Universal Robots PolyScope program: open.urp

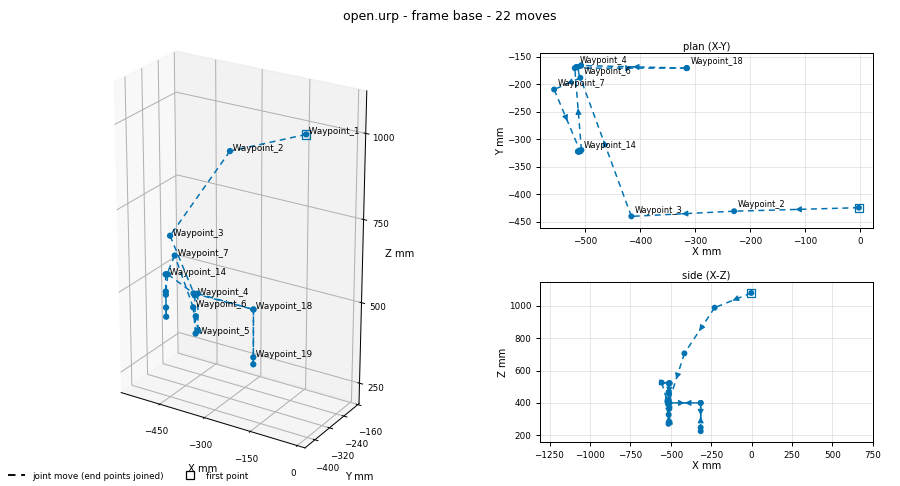
[picture p0: tool path of open.urp in frame base, 22 of 22 moves have a stored position in this frame; points joined in program order, loops and branches not executed]
Program open (installation=default directory=/programs/PrakjoyShi_Beer createdIn=5.12.6.1102099 lastSavedIn=5.12.6.1102099 robotSerialNumber=20215500597)
Calibrated DH parameters: a=[0.000193, -0.066673, -0.391568, -0.000012, 0.00005, 0]; d=[0.162643, -472.05677, 465.132521, 7.058239, 0.099746, 0.099582]; alpha=[1.571116, 0.00089, 0.003862, 1.569269, -1.569248, 0]; deltaTheta=[0, -1.413394, 7.628392, 0.068187, 0, -0.000001]
Robot Program (runOnlyOnce=true)
  MoveJ speed 60 deg/s, acceleration 80 deg/s^2 (useActiveTCP=true) feature=Base
    Waypoint Waypoint_1: TCP in base x=-1.583 y=-424.817 z=1080.554 mm, rx=-0.0045 ry=-2.2185 rz=2.2204 rad; joints [0.002, -89.999, 0.003, -90.001, -0.003, 0.002] deg; TCP offset x=0 y=0 z=191.5 mm, rx=0 ry=0 rz=0 rad
    Waypoint Waypoint_2: TCP in base x=-228.579 y=-431.222 z=989.425 mm, rx=0.1477 ry=-2.1757 rz=2.1747 rad; joints [1.493, -89.92, 39.368, -135.847, 0.07, 0.005] deg
    Waypoint Waypoint_3: TCP in base x=-415.572 y=-440.598 z=706.538 mm, rx=0.0374 ry=2.1727 rz=-2.163 rad; joints [2.063, -85.755, 82.589, -172.267, 0.054, -0.516] deg
    Waypoint Waypoint_4: TCP in base x=-515.642 y=-168.639 z=393.174 mm, rx=-2.1836 ry=-2.2574 rz=0.0027 rad; joints [3.827, -83.832, 69.203, -75.39, -89.793, 1.925] deg
    URCap Gripper Activate (Robotiq_Grippers, Robotiq Inc.) dataModel(ResetAndActivateKey=false)
    URCap Gripper (Robotiq_Grippers, Robotiq Inc.) dataModel(position=0.0, force=63.92156862745098, speed=100.0, positionInDouble=0.0, forceInDouble=63.92156862745098, speedInDouble=100.0, slaveIds=[9], blocking=true)
    Waypoint Waypoint_5: TCP in base x=-513.995 y=-168.756 z=271.062 mm, rx=-2.1837 ry=-2.2577 rz=0.0027 rad; joints [3.824, -85.645, 89.178, -93.541, -89.77, 1.988] deg
  URCap Gripper (Robotiq_Grippers, Robotiq Inc.) dataModel(position=38.0, force=100.0, speed=100.0, positionInDouble=38.0, forceInDouble=100.0, speedInDouble=100.0, slaveIds=[9], blocking=true)
  MoveJ speed 60 deg/s, acceleration 80 deg/s^2 (useActiveTCP=true) feature=Base
    Waypoint Waypoint_6: TCP in base x=-508.355 y=-188.557 z=365.162 mm, rx=2.1753 ry=2.2666 rz=0 rad; joints [6.069, -84.648, 74.27, -79.533, -89.815, 3.731] deg
    Waypoint Waypoint_7: TCP in base x=-556.081 y=-209.772 z=525.944 mm, rx=-2.4486 ry=-1.9682 rz=0.0001 rad; joints [7.701, -60.708, 14.386, -43.591, -89.88, 20.001] deg
    Waypoint Waypoint_14: TCP in base x=-508.478 y=-322.557 z=521.579 mm, rx=-2.2014 ry=-2.2234 rz=0.0401 rad; joints [19.595, -63.115, 20.022, -48.453, -89.874, 18.926] deg
    Waypoint Waypoint_15: TCP in base x=-512.267 y=-322.567 z=521.57 mm, rx=-2.2014 ry=-2.2234 rz=0.0401 rad; joints [19.472, -62.139, 18.378, -47.783, -89.873, 18.801] deg
    Waypoint Waypoint_11: TCP in base x=-512.289 y=-322.554 z=458.084 mm, rx=-2.2014 ry=-2.2234 rz=0.0402 rad; joints [19.456, -71.678, 44.329, -64.2, -89.837, 18.84] deg
    Waypoint Waypoint_16: TCP in base x=-512.283 y=-322.575 z=417.932 mm, rx=-2.2013 ry=-2.2234 rz=0.0402 rad; joints [19.451, -74.525, 54.555, -71.58, -89.828, 18.862] deg
    Waypoint Waypoint_8: TCP in base x=-512.296 y=-322.578 z=389.017 mm, rx=-2.2014 ry=-2.2233 rz=0.0403 rad; joints [19.444, -75.91, 60.769, -76.41, -89.819, 18.877] deg
    Waypoint Waypoint_17: TCP in base x=-512.289 y=-322.57 z=468.034 mm, rx=-2.2014 ry=-2.2234 rz=0.0402 rad; joints [19.46, -70.742, 41.373, -62.179, -89.843, 18.837] deg
    Waypoint Waypoint_9: TCP in base x=-506.421 y=-319.932 z=522.217 mm, rx=-2.188 ry=-2.2544 rz=0.0003 rad; joints [19.417, -60.379, 14.59, -44.133, -89.874, 17.591] deg; TCP offset x=0 y=0 z=191.5 mm, rx=0 ry=0 rz=0 rad
    Waypoint Waypoint_10: TCP in base x=-518.545 y=-170.891 z=400.25 mm, rx=2.2171 ry=2.2233 rz=-0.0042 rad; joints [3.97, -83.045, 67.23, -74.144, -89.646, 3.807] deg; TCP offset x=0 y=0 z=191.5 mm, rx=0 ry=0 rz=0 rad
    Waypoint Waypoint_18: TCP in base x=-314.832 y=-170.884 z=400.234 mm, rx=2.2171 ry=2.2233 rz=-0.0041 rad; joints [6.401, -109.126, 90.204, -71.044, -89.654, 6.252] deg
    Waypoint Waypoint_19: TCP in base x=-314.834 y=-170.918 z=247.923 mm, rx=2.217 ry=2.2233 rz=-0.0042 rad; joints [6.362, -112.11, 114.622, -92.479, -89.633, 6.291] deg
    Waypoint Waypoint_20: TCP in base x=-314.83 y=-170.903 z=225.152 mm, rx=2.217 ry=2.2233 rz=-0.0043 rad; joints [6.354, -111.859, 117.807, -95.918, -89.633, 6.297] deg
    Waypoint Waypoint_21: TCP in base x=-314.817 y=-170.895 z=400.233 mm, rx=2.217 ry=2.2233 rz=-0.0042 rad; joints [6.402, -109.128, 90.206, -71.044, -89.652, 6.249] deg
    Waypoint Waypoint_22: TCP in base x=-507.066 y=-166.173 z=400.326 mm, rx=2.2169 ry=2.2235 rz=-0.0044 rad; joints [3.531, -84.832, 69.22, -74.352, -89.639, 3.362] deg
    Waypoint Waypoint_12: TCP in base x=-507.06 y=-166.154 z=280.804 mm, rx=2.2169 ry=2.2236 rz=-0.0044 rad; joints [3.51, -86.736, 88.913, -92.143, -89.632, 3.408] deg
    URCap Gripper (Robotiq_Grippers, Robotiq Inc.) dataModel(position=0.0, force=63.92156862745098, speed=100.0, positionInDouble=0.0, forceInDouble=63.92156862745098, speedInDouble=100.0, slaveIds=[9], blocking=true)
    Waypoint Waypoint_13: TCP in base x=-513.008 y=-168.7 z=327.506 mm, rx=-2.1022 ry=-2.3346 rz=0 rad; joints [3.858, -85.632, 80.893, -85.173, -89.814, -2.097] deg
